// TIA Portal V17 export
// export: Created 2025-11-19T10:30:00.000Z, ExportSetting WithDefaults, DisplayName Totally Integrated Automation Portal, DisplayVersion V17
ORGANIZATION_BLOCK "Main"   // OB1, LAD, ProgramCycle
{ S7_Optimized_Access := 'TRUE' }
VERSION : 0.1
// stored: AutoNumber true, IsIECCheckEnabled false
   VAR_INPUT
      Initial_Call : Bool;
      Remanence : Bool;
   END_VAR
BEGIN

REGION Network 1: Motor Control Logic - BUGGY
   // BUG 1: Missing negation on Start contact - motor stays on permanently once started (latching error)
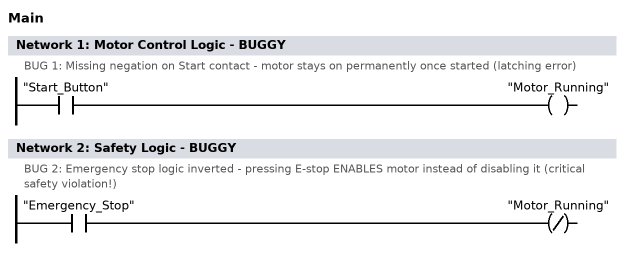
   RUNG wire#powerrail
      Contact( "Start_Button" )
      Coil( "Motor_Running" )
   END_RUNG
   // the same network as SCL:
   "Motor_Running" := "Start_Button";
END_REGION

REGION Network 2: Safety Logic - BUGGY
   // BUG 2: Emergency stop logic inverted - pressing E-stop ENABLES motor instead of disabling it (critical safety violation!)
   RUNG wire#powerrail
      Contact( "Emergency_Stop" )
      I_Coil( "Motor_Running" )
   END_RUNG
   // the same network as SCL:
   "Motor_Running" := NOT "Emergency_Stop";
END_REGION
END_ORGANIZATION_BLOCK
